PROGRAM MAIN
VAR
DPAD		: FB_BA_CarelessDPAD := (
					aIdentifier := [
	(* Level 1 *)		(	eNodeType:=E_BA_NodeType.eBuilding,			sSeparator_ObjectName := '-', 	sSeparator_Description := ' - ',	nIndexDigits := 0),
	(* Level 2 *)		(	eNodeType:=E_BA_NodeType.eFloor,			sSeparator_ObjectName := '-', 	sSeparator_Description := ' - ',	nIndexDigits := 0),
	(* Level 3 *)		(	eNodeType:=E_BA_NodeType.eTrade,			sSeparator_ObjectName := '-', 	sSeparator_Description := ' - ',	nIndexDigits := 0),
	(* Level 4 *)		(	eNodeType:=E_BA_NodeType.ePlant,			sSeparator_ObjectName := '-', 	sSeparator_Description := ' - ',	nIndexDigits := 2),
	(* Level 5 *)		(	eNodeType:=E_BA_NodeType.eAggregate,		sSeparator_ObjectName := '-', 	sSeparator_Description := ' - ',	nIndexDigits := 2),
	(* Level 6 *)		(	eNodeType:=E_BA_NodeType.eFunction,			sSeparator_ObjectName := '-', 	sSeparator_Description := ' - ',	nIndexDigits := 2)
					]
				);
//	Level 1 Gebäude 	
//	Level 1 Building 	
		B			: FB_BA_View := (
						sObjectName		:= 'B',	
						sDescription	:= 'Building B',	
						eDPADMode		:= E_BA_DPADMode.eInclude					
					);
// Level 2 Gebäudeteil
// Level 2 Part of building						
			PB1			: FB_BA_View := (
							iParent 		:= B,
							sObjectName		:= '{PB1}',		
							sDescription	:= '{Part of building 1}',
							eDPADMode		:= E_BA_DPADMode.eInclude					
						);   
// Level 3 Gewerk Automationsschwerpunkt
// Level 3 Trade AutomationFocalPoint                                                                                       	
				ACE			: FB_BA_AutomationControl := (
								iParent 		:= PB1,
								sObjectName		:= '{ACE}',
								sDescription	:= '{Automation Control}',			
								eDPADMode		:= E_BA_DPADMode.eInclude					
							);
// Level 3 Gewerk Gebäudeautomation Allgemein	- SERVER
// Level 3 Trade building automation general	- SERVER                                                                       	
				BAG			: FB_BA_BuildingAutomationServer := (
								iParent 		:= PB1,
								sObjectName		:= '{BAG}',
								sDescription	:= '{Building Automation}',			
								eDPADMode		:= E_BA_DPADMode.eInclude
							);    	
// Level 3 Gewerk Wärmeversorgungsanlagen  
// Level 3 Trade Heat supply systems, heat distribution  --> 	HD = heat distribution, HG = heat generation
				HTG			: FB_BA_Heating := (
								iParent 		:= PB1,
								sObjectName		:= '{HTG}',
								sDescription	:= '{Heating}',        		
								eDPADMode		:= E_BA_DPADMode.eInclude			
							);     	    
// Level 3 Gewerk Luftechnische Anlagen      
// Level 3 Trade ventilation system        
				ACS			: FB_BA_AirConditioning := (
								iParent 		:= PB1,
								sObjectName		:= '{ACS}',
								sDescription	:= '{Air Conditioning}',  									
								eDPADMode		:= E_BA_DPADMode.eInclude					
							);  			     
// Level 3 Gewerk Raumautomation	- SERVER
// Level 3 Trade room automation	- SERVER
				ROM			: FB_BA_RoomAutomationServer := (
								iParent			:= PB1,
								sObjectName		:= '{ROM}',
								sDescription	:= '{Room automation}',        											
								eDPADMode		:= E_BA_DPADMode.eInclude
							);
// Level 3 Gewerk Gefahrenmelde- und Alarmanlagen   
// Level 3 Trade Hazard Detection and Alarm Systems  				
				HDAS		: FB_BA_HazardDetectionAlarmSystems:= (
								iParent 		:= PB1,
								sObjectName		:= '{GMA}',
								sDescription	:= '{Hazard detection and alarm systems}',			
								eDPADMode		:= E_BA_DPADMode.eInclude
							);
// Level 3 Gewerk Türen, Tore, Fenster, Sonnenschutz	- SERVER
// Level 3 Trade Doors, gates, windwos, sun protection	- SERVER
				DGWSP		: FB_BA_DGWSPServer := (
								iParent 		:= PB1,
								sObjectName		:= '{TTF}',
								sDescription	:= '{Doors - gates - windows - sun-protection}',			
								eDPADMode		:= E_BA_DPADMode.eInclude
							);								
// SystemTime Settings								
	BACnetTime_TO_SysTime		: FB_BA_BACnetTime_TO_SysTime;	
	ExternalSysTime				: FB_BA_ExternalSysTime;
END_VAR

//	Level 1 Gebäude 	Building		
	B();
// Level 2 Gebäudeteil		Part of building
		PB1();
// Level 3 Gewerk Automation							Trade Automation			
			ACE(); 							
// Level 3 Gewerk Gebäudeautomation Allgemein			Trade BuildingAutomationGeneral			
			BAG(); 								
// Level 3 Gewerk Wärmeversorgungsanlagen				Trade Heat supply systems	
			HTG(); 	
// Level 3 Gewerk Lufttechnische Anlagen				Trade ventilation system	
			ACS(); 								
// Level 3 Gewerk Raumautomation						Trade room automation 
			ROM(); 		
// Level 3 Gewerk Gefahrenmelde- und Alarmanlagen		Trade Hazard detection and alarm systems
			HDAS();	
// Level 3 Gewerk Türen, Tore, Fenster, Sonnenschutz	Trade Doors, gates, windows, sun protection			
			DGWSP();	

//	BACnetTime_TO_SysTime();	
	ExternalSysTime();

END_PROGRAM

(* stored: Version 1.1.0.1, ProductVersion 3.1.4024.13
   POU MAIN: Id {992dd72a-c6fb-4b96-9f6e-3c624331df19}, SpecialFunc None *)
